{attribute 'qualified_only'}
VAR_GLOBAL
	
Motor1 : FB_Motor;
Motor2 : FB_Motor;

PopupTest1 : FB_TestPopup;
PopupTest2 : FB_TestPopup;


MX2_UDTs_Check : _3G3AX_MX2_ECT_A841956B;
MX2_Outputs : MX2_Outputs;


END_VAR

VAR_GLOBAL PERSISTENT
    nCycleCount : DINT := 0; 
    fTargetTemperature : REAL := 25.5;
    bMachineFault : BOOL := FALSE;
END_VAR

(* stored: Version 1.1.0.1, ProductVersion 3.1.4026.18
   GVL GVL: Id {7f66a5fd-75bd-49a5-970e-b53ba6bb8e01} *)
